PROGRAM MAIN
VAR
END_VAR

FlyingSaw(); //we call the program

END_PROGRAM

(* stored: Version 1.1.0.1, ProductVersion 3.1.4024.12
   POU MAIN: Id {69eac508-d6c0-492e-a31a-0761a161e4e8}, SpecialFunc None *)
